// Name and initial range of the arrays cannot be change.
// Name of GVL file also cannot be change.
// More information in documentation on infosys.beckhoff.com.
{attribute 'qualified_only'}
VAR_GLOBAL
	mb_Input_Coils AT%I*						: ARRAY [0..99] OF BOOL;			// Slave TCP digital inputs (max [0..255] OF BOOL)
	mb_Output_Coils AT%Q*						: ARRAY [0..99] OF BOOL;			// Slave TCP digital outputs (max [0..255] OF BOOL)
	mb_Input_Registers AT%I*					: ARRAY [0..99] OF WORD;			// Slave TCP input registers (max [0..255] OF WORD)
	mb_Output_Registers AT%Q*					: ARRAY [0..99] OF WORD;			// Slave TCP output registers (max [0..255] OF WORD)	
END_VAR

(* stored: Version 1.1.0.1, ProductVersion 3.1.4024.15
   GVL GVL_ModbusTCP_Server: Id {56b7a77e-e858-46a4-89c7-7358de00c226} *)
